(* PLC project Tc2_Utilities.BYTEARR_TO_MAXSTRING Demo, tc3-libraries-kb TwinCAT 3.1 *)
(* stored: creationDateTime 2026-05-10T19:00:00, modificationDateTime 2026-05-10T19:00:00 *)

PROGRAM P_Demo_BYTEARR_TO_MAXSTRING
  VAR
    rResult : T_MaxString;  (* BYTEARR_TO_MAXSTRING 返回值 *)
    bRun : BOOL;  (* 触发一次调用 *)
    ar : ARRAY[0..MAX_STRING_LENGTH] OF BYTE;  (* 测试用本地变量 *)
  END_VAR

            // ============================================================
// Tc2_Utilities.BYTEARR_TO_MAXSTRING 演示程序（FUNCTION）
// ============================================================
// 验证步骤：
//   1. 引用 Tc2_Utilities
//   2. 编译 + 登录
//   3. 强制 bRun := TRUE 一个周期
//   4. 在线监视 rResult / 各 demo 变量
// ============================================================

ar[0] := 16#48; ar[1] := 16#69;
IF bRun THEN
    rResult := BYTEARR_TO_MAXSTRING(ar);
    bRun := FALSE;
END_IF;

          
END_PROGRAM
